# EPICS substitutions: 2024-07-04/TEST-DI-IOC-01/TEST-DI-IOC-01App/Db/TEST-DI-IOC-01_expanded.substitutions
# This file was automatically generated on Fri 05 Jul 2024 17:42:33 BST from
# source: /dls_sw/work/R3.14.12.7/support/GIGE-BUILDER/etc/makeIocs/TEST-DI-IOC-01.xml
#
# *** Please do not edit this file: edit the source file instead. ***
#

# Macros:
#  P        Device Prefix
#  R        Device Suffix
#  PORT     Asyn Port name
#  TIMEOUT  Timeout
#  ADDR     Asyn Port address
file $(ADSIMDETECTOR)/db/simDetector.template
{
pattern { P, R, PORT, TIMEOUT, ADDR }
    { "TEST-AD-SIM-01", ":CAM:", "ADSIM.CAM", "1", "0" }
}

# Macros:
#  P             Device Prefix
#  R             Device Suffix
#  PORT          Asyn Port name
#  TIMEOUT       Timeout
#  ADDR          Asyn Port address
#  NDARRAY_PORT  Input Array Port
#  NDARRAY_ADDR  Input Array Address
#  ENABLED       Plugin Enabled at startup?
#  SCANRATE      Specified scan rate for cpu intensive PVs
file $(ADCORE)/db/NDProcess.template
{
pattern { P, R, PORT, TIMEOUT, ADDR, NDARRAY_PORT, NDARRAY_ADDR, ENABLED, SCANRATE }
    { "TEST-AD-SIM-01", ":PROC:", "ADSIM.PROC", "1", "0", "ADSIM.CAM", "0", "1", "I/O Intr" }
}

# Macros:
#  P             Device Prefix
#  R             Device Suffix
#  PORT          Asyn Port name
#  TIMEOUT       Timeout
#  ADDR          Asyn Port address
#  NDARRAY_PORT  Input Array Port
#  NDARRAY_ADDR  Input Array Address
#  ENABLED       Plugin Enabled at startup?
#  SCANRATE      Specified scan rate for cpu intensive PVs
file $(ADCORE)/db/NDROI.template
{
pattern { P, R, PORT, TIMEOUT, ADDR, NDARRAY_PORT, NDARRAY_ADDR, ENABLED, SCANRATE }
    { "TEST-AD-SIM-01", ":ROI:", "ADSIM.ROI", "1", "0", "ADSIM.CAM", "0", "1", "I/O Intr" }
}

# Macros:
#  P             Device Prefix
#  R             Device Suffix
#  PORT          Asyn Port name
#  TIMEOUT       Timeout
#  ADDR          Asyn Port address
#  NDARRAY_PORT  Input Array Port
#  NDARRAY_ADDR  Input Array Address
#  ENABLED       Plugin Enabled at startup?
#  SCANRATE      Specified scan rate for cpu intensive PVs
file $(ADCORE)/db/NDTransform.template
{
pattern { P, R, PORT, TIMEOUT, ADDR, NDARRAY_PORT, NDARRAY_ADDR, ENABLED, SCANRATE }
    { "TEST-AD-SIM-01", ":TR:", "ADSIM.TR", "1", "0", "ADSIM.CAM", "0", "1", "I/O Intr" }
}
